// TIA Portal V20 export
TYPE "typeIntConditionHmiInterface"
// stored: Access Published, Namespace Unit1.Em8
   STRUCT
      Axis_17 { S7_SetPoint := 'True'} : "LER_typeAxisIntlockAll";   // AnodeMainPnP1AxisX
      Actuator_50 { S7_SetPoint := 'True'} : "LER_typeAxisActuatorCondition";   // AnodeNgBoxLockUpDown
      Actuator_51 { S7_SetPoint := 'True'} : "LER_typeAxisActuatorCondition";   // AnodeMaintenanceMovingFixFrontFwdBwd
      Actuator_52 { S7_SetPoint := 'True'} : "LER_typeAxisActuatorCondition";   // AnodeMaintenanceMovingFixFrontFwdBwd
      Actuator_53 { S7_SetPoint := 'True'} : "LER_typeAxisActuatorCondition";   // AnodeMaintenanceMovingFixFrontFwdBwd
      Actuator_54 { S7_SetPoint := 'True'} : "LER_typeAxisActuatorCondition";   // AnodeMaintenanceMovingFixFrontFwdBwd
      Actuator_55 { S7_SetPoint := 'True'} : "LER_typeAxisActuatorCondition";   // AnodeMaintenanceMovingFixFrontFwdBwd
   END_STRUCT;
END_TYPE
